// TwinCAT 3 PLC project CX8190_OPC_UA_Client
// ProgramVersion: 3.1.4023.0
// libraries:
//   Tc2_Standard, * (Beckhoff Automation GmbH)
//   Tc2_System, * (Beckhoff Automation GmbH)
//   Tc3_Module, * (Beckhoff Automation GmbH)
// project tree:
//   / PlcTask.TcTTO
//   POUs/ MAIN.TcPOU

CONFIGURATION CX8190_OPC_UA_Client
    RESOURCE PLC ON TwinCAT3
        TASK PlcTask(INTERVAL := T#10ms, PRIORITY := 20);
        PROGRAM MAIN WITH PlcTask : MAIN;
    END_RESOURCE
END_CONFIGURATION

// ---- POUs/MAIN.TcPOU
PROGRAM MAIN
VAR
	Timer_On_Delay: TON;
	Start: BOOL;
	QTY: INT;
END_VAR

Timer_On_Delay(IN:= Start XOR Timer_On_Delay.Q,PT:=T#1S,Q=>);
IF(Timer_On_Delay.Q)
	THEN
	//QTY++;
	//QTY+=1;
	QTY:= QTY+1;
END_IF

END_PROGRAM
